TYPE FB_Interpolation_Hand :
STRUCT
	Y_pos : BOOL;
	Y_neg : BOOL;
	X_pos : BOOL;
	X_neg : BOOL;
END_STRUCT
END_TYPE

(* stored: Version 1.1.0.1, ProductVersion 3.1.4018.5
   DUT FB_Interpolation_Hand: Id {176aa8f8-36f6-40a6-879a-ca5aec7f2398} *)
